(* PLC project st_project, plcc plcc tests 1 *)
(* stored: creationDateTime 2026-09-27T00:00:00 *)

TYPE Mode : (Idle, Running, Fault);
END_TYPE

TYPE Percent : INT(0..100);
END_TYPE

TYPE Counts : ARRAY[1..4] OF DINT;
END_TYPE

TYPE Speed : REAL;
END_TYPE

TYPE Motor : STRUCT
  speed : Speed;
  starts : UDINT := 7;
  label : STRING(16);
END_STRUCT;
END_TYPE

FUNCTION Clamp : INT
  VAR_INPUT
    v : INT;
    hi : INT;
  END_VAR

            
IF v > hi THEN
    Clamp := hi;
ELSE
    Clamp := v;
END_IF;

          
END_FUNCTION

FUNCTION_BLOCK Accumulator
  VAR_INPUT
    add : DINT;
  END_VAR
  VAR_OUTPUT
    total : DINT;
  END_VAR

            total := total + add; (* entities: a < b && c *)
          
END_FUNCTION_BLOCK

PROGRAM Main
  VAR
    start AT %IX0.0 : BOOL;
    raw AT %IW1 : INT;
    running AT %QX0.1 : BOOL;
    level AT %QW1 : INT;
  END_VAR
  VAR
    mode : INT;
    pct : Percent := 42;
    hist : Counts := [2(10), 20, 30];
    m : Motor;
    acc : Accumulator;
    scans : DINT;
    histsum : DINT;
  END_VAR
  VAR CONSTANT
    LIMIT_HI : INT := 1000;
  END_VAR
  VAR RETAIN
    boots : UDINT;
  END_VAR

            
scans := scans + 1;
IF start THEN
    mode := 1;
ELSE
    mode := 0;
END_IF;
running := mode = 1;
level := Clamp(v := raw * 2, hi := LIMIT_HI);
acc(add := 1);
histsum := hist[1] + hist[2] + hist[3] + hist[4] + INT_TO_DINT(pct);
m.starts := m.starts + 1;

          
END_PROGRAM

CONFIGURATION Plant
  RESOURCE Cpu ON PLC
    TASK Fast(INTERVAL := T#10ms, PRIORITY := 1);
    PROGRAM main1 WITH Fast : Main;
  END_RESOURCE
END_CONFIGURATION
